TYPE T_CodePRODUCEDATE : STRING[14];
END_TYPE

(* stored: Version 1.1.0.1, ProductVersion 3.1.4024.15
   DUT T_CodePRODUCEDATE: Id {79b9e02c-75c9-4914-ab3a-b3d252985250} *)
